// TIA Portal V19 export
FUNCTION_BLOCK "TYPIC_C701_IF_VEKR"   // FB96, FBD
TITLE = TYPIC_C701_IF_VEKR: Verwarmingskring
{ S7_Optimized_Access := 'TRUE' }
AUTHOR : OCOTECH
FAMILY : Typical
NAME : C701.711
// Logisch Object Besturing: C701.711
// 
// 								De interne functie Verwarmingskring verzorgt de interne besturing,
// 								bewaking en fysieke aansturing van een collectorkring behorend tot
// 								de klimaatinstallatie.
// 								Er wordt een vrijgave aan de pompen gegeven als er een warmtevraag
// 								is. De drukregeling gebeurt door de pomp zelf. Antioblokkeer
// 								beveiliging is ook instelbaar op de pomp zelf.
// 								De collector verwarming bestaat uit 2 kringen:
// 								Kring verwarmingsbatterijen
// 								Kring ventiloconvectoren en klimaatkasten
// stored: MemoryReserve 10, SetENOAutomatically false
   VAR_INPUT
      STU_IF_VEKR { ExternalAccessible := 'False'; ExternalVisible := 'False'; ExternalWritable := 'False'} : Bool;   // Sturing van de interne functie klimaatregeling (IF), warmtevraag voor kring
      IN_AAN_PMP { ExternalAccessible := 'False'; ExternalVisible := 'False'; ExternalWritable := 'False'} : Bool;   // Terugmelding aansturing pomp (1 = Aan)
      IN_THM { ExternalAccessible := 'False'; ExternalVisible := 'False'; ExternalWritable := 'False'} : Bool;   // Status thermische beveiliging (1 = OK)
      IN_DME { ExternalAccessible := 'False'; ExternalVisible := 'False'; ExternalWritable := 'False'} : Real;   // Drukmeting
      IN_TME_IN { ExternalAccessible := 'False'; ExternalVisible := 'False'; ExternalWritable := 'False'} : Real;   // Temperatuur vertrek
      IN_TME_UIT { ExternalAccessible := 'False'; ExternalVisible := 'False'; ExternalWritable := 'False'} : Real;   // Temperatuur retour
      CFG_TYD_FB { ExternalAccessible := 'False'; ExternalVisible := 'False'; ExternalWritable := 'False'} : Time;   // Vertragingstijd storing foute terugmelding
   END_VAR
   VAR_OUTPUT
      VAR_IF_VEKR { ExternalAccessible := 'False'; ExternalVisible := 'False'; ExternalWritable := 'False'} : "C701_VAR_IF_VEKR_TYPIC";   // Struct met alle variabelen naar bovenliggende functies
      OUT_VGV { ExternalAccessible := 'False'; ExternalVisible := 'False'; ExternalWritable := 'False'} : Bool;   // Vrijgave pomp
   END_VAR
   VAR_IN_OUT
      STU_VGV_VEKR_AAN : Bool;   // Vrijgave inschakelen NIET NODIG?
   END_VAR
   VAR
      STO { ExternalWritable := 'False'} : Struct   // Storingen
         A001 : Bool;   // Storing van de motorbeveiliging van de pomp
         A002 : Bool;   // Fout temperatuurmeting vertrek
         A003 : Bool;   // Fout temperatuurmeting retour
         A004 : Bool;   // Fout drukmeting
         M001 : Bool;   // De motor is afgekoppeld via de werkschakelaar
      END_STRUCT;
      VAR { ExternalWritable := 'False'} : Struct   // Variabelen
         TME_IN : Real;   // Temperatuur vertrek
         TME_UIT : Real;   // Temperatuur retour
         DME : Real;   // Druk vertrek
         VGV : Bool;   // Vrijgave voor pomp
         TYD_TOT_AAN : LInt;   // Totaal aantal draaiuren (in seconden)
         TYD_TOT_AAN_UUR : LInt;   // Totaal aantal draaiuren (in uren)
      END_STRUCT;
   END_VAR
BEGIN

REGION Network 1: START
END_REGION

REGION Network 2: +++ Metingen +++
   // inlezen van vertrek- en retourtemperatuur.
END_REGION

REGION Network 3: +++ Storingen en meldingen +++
   // aanmaken van storingen en meldingen.
END_REGION

REGION Network 4: Storing A001: Storing van de motorbeveiliging van de pomp
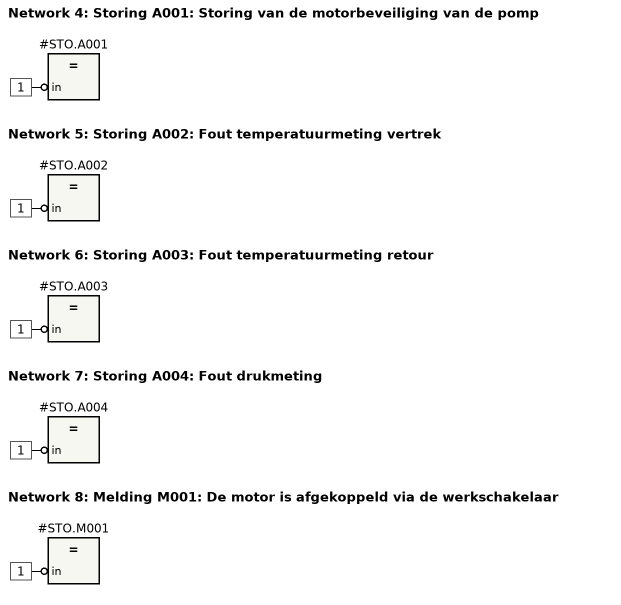
   #STO.A001 := NOT 1;
END_REGION

REGION Network 5: Storing A002: Fout temperatuurmeting vertrek
   #STO.A002 := NOT 1;
END_REGION

REGION Network 6: Storing A003: Fout temperatuurmeting retour
   #STO.A003 := NOT 1;
END_REGION

REGION Network 7: Storing A004: Fout drukmeting
   #STO.A004 := NOT 1;
END_REGION

REGION Network 8: Melding M001: De motor is afgekoppeld via de werkschakelaar
   #STO.M001 := NOT 1;
END_REGION

REGION Network 9: +++ Sturingen pomp +++
   // bij warmtevraag pomp vrijgave geven.
END_REGION

REGION Network 10: +++ Urentellers +++
   // tellen van de tijdsduur dat de motor draait.
END_REGION

REGION Network 11 (SCL): EINDE
   // Variabelen van intern scada rakvlak naar outputs copieren
   #VAR_IF_VEKR.STO := #STO;
END_REGION
END_FUNCTION_BLOCK
